(* IEC 61131-3 sources: Lasal/CPU_5344_V01/Class/AssemblyOneProdRuleV2, 1 file *)

(* ---- AssemblyOneProdRuleV2.st ---- *)
(*!
<Class
	Name               = "AssemblyOneProdRuleV2"
	Revision           = "0.0"
	RealtimeTask       = "false"
	CyclicTask         = "false"
	BackgroundTask     = "true"
	DefBackground      = "1000 ms"
	Sigmatek           = "false"
	OSInterface        = "false"
	HighPriority       = "false"
	Automatic          = "false"
	UpdateMode         = "Prescan"
	SharedCommandTable = "true"
	Objectsize         = "(480,300)">
	<Channels>
		<Server Name="Amount" Visualized="true" Initialize="false" WriteProtected="false" Retentive="false"/>
		<Server Name="ClassSvr" Visualized="false" Initialize="false" WriteProtected="true" Retentive="false"/>
		<Server Name="Length" Visualized="true" Initialize="false" WriteProtected="false" Retentive="false"/>
		<Server Name="ProductId" Visualized="true" Initialize="false" WriteProtected="false" Retentive="false"/>
		<Server Name="rnr" Visualized="true" Initialize="true" WriteProtected="false" Retentive="false"/>
		<Server Name="strDescription" Visualized="true" Remotely="true" Initialize="true" WriteProtected="false" Retentive="false" Comment="use this channel to access the string functions"/>
		<Client Name="str_Description" Required="true" Internal="true"/>
	</Channels>
	<Network Name="AssemblyOneProdRuleV2">
		<!-- List of Components in this network -->
		<Components>
			<Object
				Name       = "str_Description"
				Class      = "EditString"
				Position   = "(120,300)"
				Visualized = "true"
				Remotely   = "true">
				<Channels>
					<Server Name="Data"/>
					<Server Name="Handle"/>
					<Server Name="NewData"/>
				</Channels>
			</Object>
		</Components>
		<Comments>
		</Comments>
		<!-- List of Connections in this network -->
		<Connections>
			<Connection Source="this.str_Description" Destination="str_Description.Data"/>
			<Connection Source="this.strDescription" Destination="str_Description.Data" Vertices="(608,330),(436,390),"/>
		</Connections>
		<!-- Headerfiles -->
		<Options>
		</Options>
	</Network>
</Class>
*)
AssemblyOneProdRuleV2 : CLASS
  //Servers:
	ClassSvr 	: SvrChCmd_DINT;
	rnr 	: SvrCh_DINT;
	strDescription 	: SvrCh_UDINT;
	Amount 	: SvrCh_DINT;
	ProductId 	: SvrCh_DINT;
	Length 	: SvrCh_DINT;
  //Clients:
	str_Description 	: CltChCmd_EditString;
  //Variables:
		ptr 	: ^AssemblyDbV2::tRecipeLine;
  //Functions:

	FUNCTION VIRTUAL GLOBAL Background
		VAR_INPUT
			EAX 	: UDINT;
		END_VAR
		VAR_OUTPUT
			state (EAX) 	: UDINT;
		END_VAR;

	FUNCTION GLOBAL WritePtr
		VAR_INPUT
			iptr 	: ^AssemblyDbV2::tRecipeLine;
		END_VAR;

	FUNCTION GLOBAL WriteDescription
		VAR_INPUT
			inStr 	: gbl_datatypes::tStr20;
		END_VAR;

	FUNCTION VIRTUAL GLOBAL strDescription::Read
		VAR_OUTPUT
			output (EAX) 	: UDINT;
		END_VAR;

	FUNCTION VIRTUAL GLOBAL strDescription::Write
		VAR_INPUT
			input (EAX) 	: UDINT;
		END_VAR
		VAR_OUTPUT
			result (EAX) 	: UDINT;
		END_VAR;

	FUNCTION VIRTUAL GLOBAL Amount::Write
		VAR_INPUT
			input (EAX) 	: DINT;
		END_VAR
		VAR_OUTPUT
			result (EAX) 	: DINT;
		END_VAR;

	FUNCTION VIRTUAL GLOBAL ProductId::Write
		VAR_INPUT
			input (EAX) 	: DINT;
		END_VAR
		VAR_OUTPUT
			result (EAX) 	: DINT;
		END_VAR;

	FUNCTION VIRTUAL GLOBAL Length::Write
		VAR_INPUT
			input (EAX) 	: DINT;
		END_VAR
		VAR_OUTPUT
			result (EAX) 	: DINT;
		END_VAR;
  //Tables:
	FUNCTION @STD
		VAR_OUTPUT
			ret_code	: CONFSTATES;
		END_VAR;
	FUNCTION GLOBAL TAB @CT_;
END_CLASS;

#pragma using EditString

FUNCTION VIRTUAL GLOBAL AssemblyOneProdRuleV2::strDescription::Read
	VAR_OUTPUT
		output (EAX) 	: UDINT;
	END_VAR

	strDescription := str_Description.Data.Read();
	output := strDescription;

END_FUNCTION

FUNCTION VIRTUAL GLOBAL AssemblyOneProdRuleV2::strDescription::Write
	VAR_INPUT
		input (EAX) 	: UDINT;
	END_VAR
	VAR_OUTPUT
		result (EAX) 	: UDINT;
	END_VAR

	strDescription := input;
	result := (str_Description.Data.Write(strDescription))$UDINT;

END_FUNCTION

FUNCTION VIRTUAL GLOBAL AssemblyOneProdRuleV2::Amount::Write
	VAR_INPUT
		input (EAX) 	: DINT;
	END_VAR
	VAR_OUTPUT
		result (EAX) 	: DINT;
	END_VAR

  if ptr <> NIL then
    Amount := input;
    ptr^.amount := Amount;
    result := Amount;
  else
    result := ACCESS_DENIED;
  end_if;

END_FUNCTION

FUNCTION VIRTUAL GLOBAL AssemblyOneProdRuleV2::ProductId::Write
	VAR_INPUT
		input (EAX) 	: DINT;
	END_VAR
	VAR_OUTPUT
		result (EAX) 	: DINT;
	END_VAR

  if ptr <> NIL then
    ProductId := input;
    ptr^.productId := ProductId;
    result := ProductId;
  else
    result := ACCESS_DENIED;
  end_if;

END_FUNCTION

FUNCTION VIRTUAL GLOBAL AssemblyOneProdRuleV2::Background
	VAR_INPUT
		EAX 	: UDINT;
	END_VAR
	VAR_OUTPUT
		state (EAX) 	: UDINT;
	END_VAR
//
//  if str_Description.NewData.Read() <> 0 then
//    _memset(dest:=#ptr^.ArtikelNummer[0], usByte:=0, cntr:=sizeof(ptr^.ArtikelNummer));
//    str_Description.ReadDataOff(udOff:=0, pData:=#ptr^.ArtikelNummer[0], udMax:=sizeof(ptr^.ArtikelNummer));
//    ptrChanged^ := TRUE;
//    str_Description.NewData.Write(input:=0);
//  end_if;

	state := READY;

END_FUNCTION

FUNCTION GLOBAL AssemblyOneProdRuleV2::WritePtr
	VAR_INPUT
		iptr 	: ^AssemblyDbV2::tRecipeLine;
	END_VAR

  ptr := iptr;
  Amount := ptr^.amount;
  ProductId := ptr^.productId;
  //str_Description.WriteDataOff(udLen:=sizeof(Samenstelling::tRegel.ArtikelNummer), udOff:=0, pData:=#ptr^.ArtikelNummer[0]);

END_FUNCTION

FUNCTION GLOBAL AssemblyOneProdRuleV2::WriteDescription
	VAR_INPUT
		inStr 	: gbl_datatypes::tStr20;
	END_VAR

  str_Description.WriteDataOff(udLen:=sizeof(inStr), udOff:=0, pData:=#inStr[0]);

END_FUNCTION

FUNCTION VIRTUAL GLOBAL AssemblyOneProdRuleV2::Length::Write
	VAR_INPUT
		input (EAX) 	: DINT;
	END_VAR
	VAR_OUTPUT
		result (EAX) 	: DINT;
	END_VAR

	Length := input;
	result := Length;

END_FUNCTION
